// TIA Portal V16 export
// export: Created 2023-02-01T15:24:13.3591852Z, ExportSetting WithDefaults, DisplayName Totally Integrated Automation Portal, DisplayVersion V16 Update 3, DisplayName TIA Portal Version Control Interface, DisplayVersion V16 Update 2, DisplayName TIA Portal Openness, DisplayVersion V16 Update 3, DisplayName STEP 7 Professional, DisplayVersion V16 Update 3, DisplayName STEP 7 Safety, DisplayVersion V16, DisplayName WinCC Professional, DisplayVersion V16 Update 3
FUNCTION "FC11101_StdDevValveBi" : Void   // FC11101, LAD
TITLE = Standard Module [DEVICE DRIVER] — Bistable Valve
{ S7_Optimized_Access := 'TRUE' }
AUTHOR : M_Gledhill
FAMILY : DeviceDriver
NAME : StdDevValveBi
VERSION : 0.8
// PRACTICAL SERIES AUTOMATION LIBRARY (PAL)   —   COPYRIGHT 2020 – M. GLEDHILL (MIT LICENCE)
//                   ———— ◆ ————
// FULL ONLINE DOCUMENTATION IS AVAILABLE AT: https://practicalseries.com/2001-pal/index.html
// stored: AutoNumber false, IsIECCheckEnabled true, SetENOAutomatically false, UDAEnableTagReadback false
   VAR_INPUT
      SYS_SIGNALS : "UT21000_Dy_SysSignals";   // Common system signals — logic and timing signals
      FBK_OPEN : Bool;   // Positive open position feedback (1 = valve open, 0 = valve not open)
      FBK_CLOSED : Bool;   // Positive closed position feedback (1 = valve closed, 0 = valve not closed)
      EXT_FAULT : Bool;   // Device external fault signal (1 = fault, 0 = healthy)
      E_STOP : Bool;   // Safety (E-STOP) signal (1 = ESTOP active, 0 = healthy)
      TRIP : Bool;   // Interlock (TRIP) signal (1 = TRIP active, 0 = healthy)
      INTERLOCK : Bool;   // Interlock (INTERLOCK) signal (1 = INTERLOCK active, 0 = healthy)
      PERMISSIVE : Bool;   // Interlock (PERMISSIVE) signal (1 = PERMISSIVE active, 0 = healthy)
      STATIC_DATA : "UT11101_St_DevValveBi";   // Static data storage (UDT)
   END_VAR
   VAR_OUTPUT
      OPEN_CMD : Bool;   // Valve open signal (1 = open the valve, 0 = no action)
      CLOSE_CMD : Bool;   // Valve close signal (1 = close the valve, 0 = no action)
   END_VAR
   VAR_IN_OUT
      DYNAMIC_DATA : "UT31101_Dy_DevValveBi";   // Dynamic data storage (UDT)
   END_VAR
   VAR_TEMP
      revInfo : "UT01000_St_SysRevision";   // Revision information for this block
      licInfo : "UT01001_St_SysLicence";   // Licensing information for this block
      calClosedElapsedTime : Real;   // Calculation - Derived closed signal elapsed time limit
      calOpenElapsedTime : Real;   // Calculation - Derived open signal elapsed time limit
      wrkOpen : Bool;   // Working - open position feedback signal (actual or derived)
      wrkClosed : Bool;   // Working - closed position feedback signal (actual or derived)
      wrkCtrlPriority40 : Bool;   // Working - priority 40 condition controls the valve
      wrkCtrlPriority30 : Bool;   // Working - priority 30 condition controls the valve
      wrkCtrlPriority20 : Bool;   // Working - priority 20 condition controls the valve
      wrkCtrlPriority10 : Bool;   // Working - priority 10 condition controls the valve
      wrkCtrlPriority00 : Bool;   // Working - priority 00 condition controls the valve
      wrkCtrlAutManOpCl : Bool;   // Working - consolidated auto/manual open or close request
      wrkTimeFbkOpenDer : Real;   // Working - value of opening timer before derived open feedback
      wrkTimeFbkClosedDer : Real;   // Working - value of closing timer before derived closed feedback
      wrkInt : Int;   // Working - storage area (integer)
      wrkReal : Real;   // Working - storage area (Real)
      wrkDInt : DInt;   // Working - storage area (double integer)
   END_VAR
   VAR CONSTANT
      k_TIME_OP_MIN : Real := 0.21;   // Minimum value for the valve operation timer
      K_TIME_SIM_MIN : Real := 0.21;   // Minimum value for the simulation operation timer
   END_VAR
   VAR_TEMP   // added for the SCL form of the ladder/FBD networks
      _w1 : Bool;
      _w2 : Bool;
      _w3 : Bool;
   END_VAR
BEGIN

REGION Network 1: Block description — Sections 1 to 2
   // ▄▄▄▄▄▄▄▄▄▄▄▄▄▄▄▄▄▄▄▄▄▄▄▄▄▄▄▄▄▄▄▄▄  ＳＴＡＮＤＡＲＤ  ▄▄ 
   // 
   // 
   // TITLE:    DEVICE DRIVER — BISTABLE VALVE
   // 
   // 
   // ▀▀▀▀▀▀▀▀▀▀▀▀▀▀▀▀▀▀▀▀▀▀▀▀▀▀▀▀▀▀▀▀▀▀▀▀▀▀▀▀▀▀▀▀ 
   // 
   // ┌──────────────────────────────────────────┐
   // │                                          │
   // │          FC11101 — SOFTWARE MODULE DESIGN SPECIFICATION (SMDS)            │
   // │                                          │
   // │      The PDF version of the SMDS for this module is available online here:        │
   // │              https://psop.uk/pal-smds-fc11101-p               │
   // │                                          │
   // │      It is also available as part of the Project User Defined Documentation,      │
   // │      it can be accessed by selecting this module in the Project Tree          │
   // │      (on the left) and pressing SHIFT+F1                        │
   // │                                          │
   // └─────────────────────────────────────── ʷᴵᴰ⁻ᶜᵇᵃ ┘
   // 
   // FC11101_StdDevValveBi controls the operation of a bistable valve configured with either open, 
   // closed, both open and closed or no position feedback (depending on the valve type).
   // 
   // The module supports automatic and manual control and can be configured with simulation 
   // mode to allow the valve limit switch signals to be overwritten and set to follow the demand 
   // position.
   // 
   // The module can be configured to either de-energise the outputs when the valve reaches the 
   // demanded position, or maintain the outputs when position is reached.
   // 
   // The module generates fault logic for the valve that will trigger specific alarms depending on the 
   // fault in question. The alarms within this block are: 
   // 
   // 
   //    •   Failed to Open 
   // 
   //    •   Failed to Close 
   // 
   //    •   Failed while Open
   // 
   //    •   Failed while Closed
   // 
   //    •   External Fault 
   // 
   // Separate operation times for opening and closing can be defined. 
   // 
   // The valve module supports all forms of interlock, permissive and trip signals, and emergency 
   // stop signals. The module has the conditional facility to allow the operator to bypass interlocks, 
   // permissive and trip conditions.
   // 
   // Various status signals are generated for supervisory systems:
   // 
   //    •   Closed
   // 
   //    •   Closing
   // 
   //    •   Open
   // 
   //    •   Opening
   // 
   //    •   Fault
   // 
   // The module also generates status signals for the selected operating modes and conditions.
   // 
   // 
   // 
   // ▄▄▄▄▄▄▄▄▄▄▄▄▄▄▄▄▄▄▄▄▄▄▄▄▄▄▄▄▄▄▄▄▄▄▄▄▄▄▄▄▄▄▄▄
   // 1.     BLOCK TECHNICAL SUMMARY
   // 
   // 
   //  ――――――――――――――――――――――――――――――――――――――――――
   //  NOMENCLATURE & ADDRESSING
   //  ――――――――――――――――――――――――――――――――――――――――――
   //  BLOCK TITLE         Bistable Valve
   //  BLOCK FUNCTION GROUP    Device Driver 
   //  BLOCK ADDRESS       FC11101
   //  BLOCK SYMBOL        FC11101_StdDevValveBi
   //  BLOCK USER ID         StdDevValveBi
   // 
   //  ――――――――――――――――――――――――――――――――――――――――――
   //  BLOCK TYPE & USAGE
   //  ――――――――――――――――――――――――――――――――――――――――――
   //  BLOCK TYPE         Function (FC)
   //  BLOCK NUMBER        11101
   //  LANGUAGE           LAD
   //  OPTIMISED ACCESS     Yes
   //  PAL USAGE TYPE       Standard block
   // 
   //  ――――――――――――――――――――――――――――――――――――――――――
   //  METRICS
   //  ――――――――――――――――――――――――――――――――――――――――――
   //  EXECUTION TIME       81.3 μs¹
   //  LOAD MEMORY       113.1 kB
   //  WORK MEMORY           2.5 kB  
   //  ――――――――――――――――――――――――――――――――――――――――――
   //                ¹ Measured on: CPU-1515-2PN (order no. 6ES7512-2AM02-0AB0) 
   //                             https://psop.uk/pal-ds-cpu1515
   // 
   // 
   // 
   // ▂▂▂▂▂▂▂▂▂▂▂▂▂▂▂▂▂▂▂▂▂▂▂▂▂▂▂▂▂▂▂▂▂▂▂▂▂▂▂▂▂▂▂▂
   // 1.1      Additional document references
   // 
   // 
   // Only those documents specified in OB1 (section DOCUMENT REFERENCES) are listed within this 
   // block. There are no additional document references.
   // 
   //                ━━━   ⬙⬙⬙⬙⬙⬙   ━━━
   // 
   // 
   // 
   // ▄▄▄▄▄▄▄▄▄▄▄▄▄▄▄▄▄▄▄▄▄▄▄▄▄▄▄▄▄▄▄▄▄▄▄▄▄▄▄▄▄▄▄▄
   // 2.     FUNCTIONAL DESCRIPTION
   // 
   // 
   // FC11101 is the Bistable Valve block, it is a comprehensive block designed to operate and monitor 
   // a standard bistable valve. 
   // 
   // 
   // 
   // ▂▂▂▂▂▂▂▂▂▂▂▂▂▂▂▂▂▂▂▂▂▂▂▂▂▂▂▂▂▂▂▂▂▂▂▂▂▂▂▂▂▂▂▂
   // 2.1     Defining a bistable valve
   // 
   // 
   // A bistable valve is any valve that has two signals to make it change state; it has two mutually 
   // exclusive output signals: an OPEN_CMD output that must be energised to drive the valve to the 
   // open position and a CLOSE_CMD output that must be energised to drive the valve to the closed 
   // position.
   // 
   // To open the valve the OPEN_CMD signal must be energised and the CLOSE_CMD signal 
   // deenergised. When the valve reaches the opened position, both signals will be deenergised² and 
   // the valve will remain in the opened state (it is stable in this condition and does not require any 
   // signal to maintain it in this state, if there were a power failure the valve would remain opened).
   // 
   // To close the valve the CLOSE_CMD signal must be energised and the OPEN_CMD signal 
   // deenergised. When the valve reaches the closed position, both signals will again be 
   // deenergised² and the valve will remain in the closed state (again the valve is stable in this 
   // condition and does not require any signal to maintain it in this state, if there were a power failure 
   // the valve would remain closed).
   // 
   // This is said to be a bistable device because once it is in a particular state, it does not (generally) 
   // require any signal to be energised to maintain that state.
   // 
   // ――――――――――
   // ²         The module can also be configured to maintain the appropriate output signal once 
   //      the required state is achieved (see § 3.2.1).
   // ――――――――――
   // 
   // 
   // 
   // ▂▂▂▂▂▂▂▂▂▂▂▂▂▂▂▂▂▂▂▂▂▂▂▂▂▂▂▂▂▂▂▂▂▂▂▂▂▂▂▂▂▂▂▂
   // 2.1.1     Comparison with an isolating valve
   // 
   // 
   // In many ways a bistable valve is very similar to an isolating valve (controlled by FC11001), it 
   // generally has only two states (it is either opened or closed); however, because the bistable valve 
   // is electrically driven (usually by a motor), if the driving signals are removed while the valve is in 
   // transit (say via an emergency stop being activated), the valve will simply stop in its current 
   // (intermediate) position and remain there until a driving signal is re-applied. This situation is 
   // discussed in §§ 2.3.1 and 3.4.1.
   // 
   // Additionally, because the bistable valve is stable in both the open and closed positions, the 
   // bistable valve does not have the normally open and normally closed³  types available to an 
   // isolating valve. A Bistable valve does not return to a specific state if power is removed from the 
   // actuator; it simply remains in its current state (even if this is an indeterminate state).
   // 
   // ――――――――――
   // ³         For an isolating valve, normally closed refers to a valve that is deenergised in the 
   //      closed state and will open when an energising signal is applied. A normally open 
   //      valve operates in the reverse arrangement, the valve is open in the deenergised 
   //      state and will only close when the energising signal is present. Normally open valves 
   //      are used in fail-safe applications where a power failure causes the valve to open by 
   //      default, usually to vent pressure or release some other motive force from the vessel 
   //      to which it is connected.
   // ――――――――――
   // 
   // 
   // 
   // 
   // ▂▂▂▂▂▂▂▂▂▂▂▂▂▂▂▂▂▂▂▂▂▂▂▂▂▂▂▂▂▂▂▂▂▂▂▂▂▂▂▂▂▂▂▂
   // 2.1.2     Valve operating times
   // 
   // 
   // A bistable valve, will move from its closed state to its open state when the OPEN_CMD signal is 
   // applied; this transition will occur in a specified time (the time taken will depend on the size and 
   // operating mechanism within the valve itself), this is referred to as the opening operation time.
   // 
   // Similarly, the transition from open to closed will occur when the CLOSE_CMD signal is applied, 
   // and again, this will occur in a specified time. This is referred to as the closing operation time. 
   // 
   // The opening and closing times can be different for a given valve. 
   // 
   // Collectively, the opening and closing times are referred to as the operating times (sometimes 
   // operation times) of the valve.
   // 
   // The maximum opening and closing times for a valve are generally given as part of the 
   // specification for the valve itself.
   // 
   // If a valve does not reach the required state within the specified maximum operating times, the 
   // valve is generally considered to be in a fault condition (either failed to open or failed to close 
   // depending on the action being undertaken).
   // 
   // 
   // 
   // ▂▂▂▂▂▂▂▂▂▂▂▂▂▂▂▂▂▂▂▂▂▂▂▂▂▂▂▂▂▂▂▂▂▂▂▂▂▂▂▂▂▂▂▂
   // 2.1.3     Valve position feedback arrangements
   // 
   // 
   // Bistable valves can be equipped with limit switch signals that positively identify the current 
   // position of the valve. There are four combinations of limit switches:
   // 
   //    1.  No limit switches         There is no positive indication of the current state 
   //                      of the valve, it is assumed to be in the expected 
   //                      state.
   // 
   //    2.  Closed limit switch only       Positive indication is given for the closed state 
   //                      only. The valve is assumed to be open (after a 
   //                      predetermined time) if the closed signal is 
   //                      inactive
   // 
   //    3.  Open limit switch only      Positive indication is given for the open state 
   //                      only. The valve is assumed to be closed (after a 
   //                      predetermined time) if the open signal is 
   //                      inactive.
   // 
   //    4.  Open and closed limit switches    Positive indication is given for both states. 
   //                      This allows the true state of the valve to be 
   //                      determined under all circumstances.
   // 
   // Note:    Positive indication of a valve state need not be determined by a limit switch 
   //      (though this is by far the most common arrangement), it could for example, be 
   //      determined by some process value: if a flow is detected after the opening of a valve, 
   //      for example.
   // 
   //      In practice, limit switches are the preferred mechanism for the positive indication 
   //      of a given valve state.
   // 
   // Where a limit switch is absent, the valve is assumed to have reached the correct position when 
   // the relevant operation time has counted for an adjustable percentage of its maximum operating 
   // time.
   // 
   // The valve can be configured to “run-on” for a specified time after the demanded position has been 
   // achieved (i.e. the block will maintain the driving signal for a time period after the limit switch is 
   // activated to ensure the valve is firmly in position).
   // 
   // The valve can also be configured to maintain either the OPEN_CMD signal or the CLOSE_CMD 
   // signal permanently once the valve has reached the desired position; i.e. the OPEN/CLOSE_CMD 
   // signals do not deenergise when the valve has reached the correct position. 
   // 
   // 
   // 
   // ▂▂▂▂▂▂▂▂▂▂▂▂▂▂▂▂▂▂▂▂▂▂▂▂▂▂▂▂▂▂▂▂▂▂▂▂▂▂▂▂▂▂▂▂
   // 2.2     Module operation
   // 
   // 
   // FC11101 is used to control (operate) a bistable valve, the module also monitors the various 
   // configurations of valve position feedback signals to determine if the valve is in a fault condition.
   // 
   // The module will drive the valve to the requested state by energising and deenergising two 
   // separate (mutually exclusive) digital signals (usually digital output signals), one signal to open 
   // the valve and one to close it.
   // 
   // These digital output signals can be configured to either deenergise when the valve reaches the 
   // required state (with a configurable run-on time) or to remain energised when the final state is 
   // reached.
   // 
   // If the requested state signal changes (either from closed to open, or from open to closed), the 
   // module will start either an opening operation timer (request has changed from closed to open) 
   // or a closing operation timer (request has changed from open to closed); these timers can have 
   // different values.
   // 
   // The valve will be expected to reach the requested state before the relevant operation timer 
   // expires; if it does not, the valve will enter a fault state and an appropriate alarm will be generated 
   // when the operation timer expires.
   // 
   // Once the valve has reached its requested state, the operation time will reset and the module 
   // will continue to monitor the state of the valve. 
   // 
   // If the request signal changes whilst the valve is in the process of changing state (e.g. the valve 
   // is requested to change from closed to open and whilst the opening operation timer is running, 
   // the request is changed back to closed), the running operation timer will be reset and the 
   // operation timer for the second request will start from its specified value. I.e. no allowance is 
   // made for how far the valve may have moved following the first request change.
   // 
   // If the valve is stable, in a given state (i.e. is not in the process of changing state) and the valve 
   // position signals no longer match the required state (e.g. the valve had correctly opened, but at 
   // some time after this, the open position feedback is lost), the valve will instantly generate an 
   // alarm condition.
   // 
   // 
   // 
   // ▂▂▂▂▂▂▂▂▂▂▂▂▂▂▂▂▂▂▂▂▂▂▂▂▂▂▂▂▂▂▂▂▂▂▂▂▂▂▂▂▂▂▂▂
   // 2.3     Safety and interlocks
   // 
   // 
   // The module, optionally, accommodates a single safety signal (emergency stop), and the 
   // standard arrangement of up to three interlock signals (interlock, permissive and trip) as follows:
   // 
   // 
   // 
   // ▂▂▂▂▂▂▂▂▂▂▂▂▂▂▂▂▂▂▂▂▂▂▂▂▂▂▂▂▂▂▂▂▂▂▂▂▂▂▂▂▂▂▂▂
   // 2.3.1     Safety (emergency stop) signal
   // 
   // 
   // Safety or emergency stop signals are hardwired signals that remove power from a device forcing 
   // it to a safe state. Such signals act independently of the software (the pressing of an emergency 
   // stop button will physically remove power from the affected devices).
   // 
   // In the case of a bistable valve, the removing of the power under emergency stop conditions, 
   // simply deenergises both outputs leaving the valve in its current state¹: if the valve were already 
   // open, it would remain open, similarly if the valve were closed, it would remain closed.
   // 
   // The leads to the question, what happens if an emergency stop activates when the valve is 
   // changing state? The answer is that the valve simply stops where it is in mid-transition (in some 
   // indeterminate, intermediate state between open and closed). To accommodate this condition, 
   // the active operation timer will simply pause at its elapsed value (the valve will remain in either 
   // the opening or closing state) until the emergency stop condition is removed, at this point, the 
   // operation timer will continue from its last elapsed value .
   // 
   // Note:    The resumption of the operation timer can be delayed by a recovery time, this is
   //      to allow the physical aspects of the valve itself to reset and resume operation 
   //      (e.g. to allow the valve motor to ramp to the correct speed &c.), this recovery time 
   //      is configurable.
   // 
   // The emergency stop signal passed to the module is used to allow the condition of the valve to 
   // be correctly interpreted within the software under emergency stop conditions.
   // 
   // The presence of an emergency stop signal is indicated via the block icon status signals generated 
   // by the module (see §§ 2.7 and 4.2).
   // 
   // Emergency stop signals cannot be bypassed under any circumstances (cf. interlock signals, 
   // below).
   // 
   // ――――――――――
   // ¹         This is unlike the isolating valve of FC11001; the isolating valve returns to a particular 
   //      state (either open or closed depending on the normally open/closed arrangement of 
   //      the valve). By comparison, the bistable simply stops in the condition it is in.
   // ――――――――――
   // 
   // 
   // 
   // ▂▂▂▂▂▂▂▂▂▂▂▂▂▂▂▂▂▂▂▂▂▂▂▂▂▂▂▂▂▂▂▂▂▂▂▂▂▂▂▂▂▂▂▂
   // 2.3.2     Interlock signals
   // 
   // 
   // There are three types of interlock signal:
   // 
   //    1.  Interlock
   //      A simple interlock that is active whenever a set of conditions is true; if active, it will 
   //      force the devices to a specified state.
   // 
   // 
   //    2.  Permissive
   //      Designates a specified “permitted” state for the device. A permissive interlock takes 
   //      no action if the device is in the non-permitted state, but once the device changes to 
   //      the permitted state, it will be prevented from changing back to the non-permitted state 
   //      (e.g. if the permitted state was closed and the valve was currently open when the 
   //      permissive signal activated, it would not force the valve to close, but once it was 
   //      closed, it would prevent it from re-opening).
   // 
   //    3.  Trip
   //      A latching interlock, it activates whenever a set of events are true (like an interlock), 
   //      but will not deactivate until the triggering conditions are removed and a reset signal 
   //      has been given (effectively a latching interlock); if active, it will force the device to a 
   //      specified state.
   // 
   // Note:    The trip reset signal is handled by the trip logic, the valve module will simply respond 
   //      to the presence or absence of a trip signal.
   // 
   // Each type of interlock has its own individual signal passed to the module (three signals in total).
   // 
   // Interlock signals can be optionally bypassed (effectively disabled) under specific, manually 
   // selected operations.
   // 
   // 
   // 
   // ▂▂▂▂▂▂▂▂▂▂▂▂▂▂▂▂▂▂▂▂▂▂▂▂▂▂▂▂▂▂▂▂▂▂▂▂▂▂▂▂▂▂▂▂
   // 2.3.3     Priority of safety and interlock signals
   // 
   // 
   // The presence of any interlock stop signal is indicated via the block icon status signals generated 
   // by the module (see § 4). The priority order of the various types of interlock (if more than one is 
   // active at the same time) is as follows:
   // 
   // 
   //  ――――――――――――――――――――――――――――――――――――――――――
   //  SIGNAL TYPE        PRIORITY        CAN BE BYPASSED
   //  ――――――――――――――――――――――――――――――――――――――――――
   //  Emergency Stop         High               NO
   //  Trip             ↑              YES
   //  Interlock             ↑              YES
   //  Permissive          Low               YES
   //  ――――――――――――――――――――――――――――――――――――――――――
   //  High priority signal take precedence over lower priority signals.
   // 
   // 
   // 
   // ▂▂▂▂▂▂▂▂▂▂▂▂▂▂▂▂▂▂▂▂▂▂▂▂▂▂▂▂▂▂▂▂▂▂▂▂▂▂▂▂▂▂▂▂
   // 2.4     Alarms and warnings
   // 
   // 
   // The module can generate up to five distinct alarms:
   // 
   // 
   //    1.  FAILED TO OPEN
   //      Indicates that the valve did not open when requested to do so. The alarm is generated 
   //      when the opening operation timer expires without the corresponding position feedback 
   //      activating
   // 
   //    2.  FAILED TO CLOSE
   //      Indicates that the valve did not close when requested to do so. The alarm is generated 
   //      when the closing operation timer expires without the corresponding position feedback 
   //      activating
   // 
   // 
   //    3.  FAILED WHILE OPEN
   //      Indicates that the valve opened correctly, but then at some later point, the position 
   //      feedback signals, indicating the open state of the valve, were lost.
   // 
   //    4.  FAILED WHILE CLOSED
   //      Indicates that the valve closed correctly, but then at some later point, the position 
   //      feedback signals, indicating the closed state of the valve, were lost.
   // 
   // 
   //    5.  EXTERNAL FAULT
   //      External fault is a separate (and optional) hardwired signal from the valve that 
   //      indicates the valve itself has detected a problem (e.g. a trip signal from a 
   //      motorised valve)
   // 
   // The module does not generate any warnings.
   // 
   // 
   // 
   // ▂▂▂▂▂▂▂▂▂▂▂▂▂▂▂▂▂▂▂▂▂▂▂▂▂▂▂▂▂▂▂▂▂▂▂▂▂▂▂▂▂▂▂▂
   // 2.4.1     Alarm — Failed to open/close
   // 
   // 
   // Failed to open and failed to close alarms are generated if the valve is required to change state 
   // and fails to do so within the time set by the relevant operation timer.
   // 
   // For example, if the valve were in a closed state and was requested to open, the failed to open 
   // alarm would be generated if the valve had not received positive indication that the valve was 
   // correctly open (from the valve limit switches) by the time the opening operation timer expired.
   // 
   // If the valve is not equipped with any limit switches, then there are no circumstances under 
   // which the failed to open and failed to close alarms can be generated (the valve is always 
   // assumed to operate correctly and be in the required position).
   // 
   // 
   // 
   // ▂▂▂▂▂▂▂▂▂▂▂▂▂▂▂▂▂▂▂▂▂▂▂▂▂▂▂▂▂▂▂▂▂▂▂▂▂▂▂▂▂▂▂▂
   // 2.4.2     Alarm — Failed while open/closed
   // 
   // 
   // Failed while open and failed while closed are generated if the valve is in a steady state (not in 
   // the process of changing from open to closed or vice versa) and the positive indication of the 
   // valve position changes to indicate the steady state position has changed.
   // 
   // An example would be for a normally closed valve, with both open and closed limit switches, 
   // to be in the open (energised) state, where the open limit is active and closed limit is inactive 
   // (positively indicating the valve is open). If the power to the valve failed (a blown fuse or broken 
   // wire, for example), the valve would deenergise and return to the closed state and this would be 
   // reflected in the state of the limit switches. The module, knowing nothing of the power failure, 
   // would expect the valve to still be open and would instantly generate a failed while open alarm.
   // 
   // If the valve is not equipped with any limit switches, then there are no circumstances under which 
   // the failed while open and failed while closed alarms can be generated (the valve is always 
   // assumed to operate correctly and be in the required position).
   // 
   // 
   // 
   // ▂▂▂▂▂▂▂▂▂▂▂▂▂▂▂▂▂▂▂▂▂▂▂▂▂▂▂▂▂▂▂▂▂▂▂▂▂▂▂▂▂▂▂▂
   // 2.4.3     Alarm — External fault
   // 
   // 
   // The external fault alarm is activated whenever the external fault signal provided to the module 
   // is active. The external fault signal is an optional signal that indicates that the valve itself is 
   // experiencing a problem. The signal is more commonly associated with motorised valves where 
   // thermal overload signals are used to indicate that the valve motor has experienced a fault, 
   // it could also be used to indicate the loss of pneumatic pressure for pneumatic solenoid valves.
   // 
   // 
   // 
   // ▂▂▂▂▂▂▂▂▂▂▂▂▂▂▂▂▂▂▂▂▂▂▂▂▂▂▂▂▂▂▂▂▂▂▂▂▂▂▂▂▂▂▂▂
   // 2.4.4     Resetting alarm conditions
   // 
   // 
   // The four alarms derived from valve position feedback signals:
   // 
   //    1.  FAILED TO OPEN
   // 
   //    2.  FAILED TO CLOSE
   // 
   //    3.  FAILED WHILE OPEN
   // 
   //    4.  FAILED WHILE CLOSED
   // 
   // Are latching alarms, if the alarm conditions occur, the valve will be placed in a fault condition 
   // (see § 2.5) and will no longer be operable, the valve will remain in a deenergised condition until 
   // the fault is corrected.
   // 
   // The alarm conditions are only reset when the module receives a RESET command (usually 
   // from the operator).
   // 
   // The fifth alarm:
   // 
   //    5.  EXTERNAL FAULT
   // 
   // Is a non-latching alarm that is reset automatically whenever the external fault signal is 
   // deactivated. It should be noted however, that the cause of the external fault (say a thermal 
   // overload) may itself, require some form of manual or physical reset, before the fault condition 
   // is removed.
   // 
   // 
   // 
   // ▂▂▂▂▂▂▂▂▂▂▂▂▂▂▂▂▂▂▂▂▂▂▂▂▂▂▂▂▂▂▂▂▂▂▂▂▂▂▂▂▂▂▂▂
   // 2.5     Fault conditions
   // 
   // 
   // The valve is in a fault condition if any alarm conditions is active:
   // 
   //    1.  FAILED TO OPEN
   // 
   //    2.  FAILED TO CLOSE
   // 
   //    3.  FAILED WHILE OPEN
   // 
   //    4.  FAILED WHILE CLOSED
   // 
   //    5.  EXTERNAL FAULT
   // 
   // A valve cannot operate if any fault condition is active and it will return to its deenergised state.
   // 
   // For a normally closed valve, the deenergised state is closed and for a normally open valve, 
   // the deenergised state is open.
   // 
   // A valve that is in a fault state will ignore any request that would move it to an energised state, 
   // irrespective of the source of the command: automatic operation, manual operation or even an 
   // interlock condition.
   // 
   // 
   // The valve will remain in a fault state until all alarms have been reset, in the case of the four limit 
   // switch derived alarms the module must receive a RESET command (see § 2.4.4) to remove the 
   // alarms, and consequently, the fault conditions.
   // 
   // The EXTERNAL FAULT alarm is a non-latching alarm that is reset automatically whenever the 
   // external fault signal is deactivated, consequently, the fault state will automatically reset when 
   // the external fault signal deactivates.
   // 
   // It should be noted however, that the cause of the external fault (say a thermal overload) may 
   // itself, require some form of manual or physical reset, before the fault condition is removed.
   // 
   // 
   // 
   // ▂▂▂▂▂▂▂▂▂▂▂▂▂▂▂▂▂▂▂▂▂▂▂▂▂▂▂▂▂▂▂▂▂▂▂▂▂▂▂▂▂▂▂▂
   // 2.6     Operating modes
   // 
   // 
   // The module supports the following optional modes of operation:
   // 
   //    •   Automatic/manual mode (allows the operator to take manual control of the valve 
   //      and open or close it irrespective of the control system requirements)
   // 
   //    •   Interlock bypass mode (allows the operator to override permissive, interlock and 
   //      trip signals
   // 
   //    •   Simulation mode (allows the operator to override the current instrument position 
   //      feedback signals  simulated values)
   // 
   //    •   Remote/local/all selection (allows control of the instrument to be restricted to a 
   //      specific SCADA/HMI device) 
   // 
   //    •   Faceplate disabled (informs the supervisory system not to display any faceplates 
   //      for the device, preventing graphical operator selections)
   // 
   // 
   // 
   // ▂▂▂▂▂▂▂▂▂▂▂▂▂▂▂▂▂▂▂▂▂▂▂▂▂▂▂▂▂▂▂▂▂▂▂▂▂▂▂▂▂▂▂▂
   // 2.6.1     Automatic and manual control modes
   // 
   // 
   // By default, the module will be in automatic mode; this means that any open or close instruction 
   // received by the module from the control software (continuous or sequential control) will cause 
   // the valve to adopt the requested state (if the valve is not in fault and is free of interlock and 
   // safety conditions).
   // 
   // If the module is switched to manual mode, the automatic control signals will be ignored and the 
   // module will adopt the state required by the manual request signals set by the operator 
   // (again, the valve must not be in fault and must be free of interlock and safety conditions).
   // 
   // Selecting automatic or manual mode is an operator action and can be implemented at any time. 
   // Changing from automatic mode to manual mode is a bumpless operation, in which the initial 
   // manual state of the valve is set to match the current automatic state. For example, if a valve 
   // were open under automatic control, switching the valve to manual would cause the initial 
   // manual state to be set to open (matching the automatic state), ensuring that the valve does not 
   // initially change state when changing to manual mode.
   // 
   // Once manual mode is established, the operator is free to open and close the valve as required.
   // 
   // There is no bumpless transfer back to automatic mode, the valve will simply adopt the state 
   // required by the control software.
   // 
   // Interlocks and safety signals operate in exactly the same way for a valve in manual mode 
   // as they do for a valve in automatic mode and will take priority over any command issued in either 
   // automatic or manual mode.
   // 
   // 
   // 
   // ▂▂▂▂▂▂▂▂▂▂▂▂▂▂▂▂▂▂▂▂▂▂▂▂▂▂▂▂▂▂▂▂▂▂▂▂▂▂▂▂▂▂▂▂
   // 2.6.2     Interlock bypass mode
   // 
   // 
   // Interlock bypass mode allows the three interlock types (trip, interlock and permissive) to be 
   // overridden (bypassed) by the operator.
   // 
   // If bypass mode is activated, any interlock signal will be ignored by the module.
   // 
   // Bypass mode is an entirely manual operation that can only be initiated by an operator, usually 
   // via a supervisory system (SCADA or HMI).
   // 
   // 
   // 
   // ▂▂▂▂▂▂▂▂▂▂▂▂▂▂▂▂▂▂▂▂▂▂▂▂▂▂▂▂▂▂▂▂▂▂▂▂▂▂▂▂▂▂▂▂
   // 2.6.3     Simulation mode
   // 
   // 
   // The module can be switched to a simulation mode, under which any positive position feedback 
   // signals from valve limit switches are replaced by simulated signals selected by the operator. 
   // Simulation mode can be used during testing and can also be applied in a process environment 
   // if a fault condition is detected within the valve.
   // 
   // The operator can select any one of the following possible simulation arrangements (only one 
   // can be active at any given time):
   // 
   // 
   //    •   Follow demand    The simulation will generate open and closed signals that 
   //                 match the requested state of the valve
   // 
   //    •   Open          The simulation will generate signals to give a permanently 
   //                 open state for the valve, irrespective of any valve state 
   //                 request (allows failed open conditions to be simulated)
   // 
   //    •   Closed           The simulation will generate signals to give a permanently 
   //                 closed state for the valve, irrespective of any valve state 
   //                 request (allows failed closed conditions to be simulated)
   //                 request (allows failed open conditions to be simulated)
   // 
   //    •   No limits       No position feedback signals will be simulated
   // 
   // Simulation mode is a manual operation that can only be initiated by an operator.
   // 
   // 
   // 
   // ▁▁▁▁▁▁▁▁▁▁▁▁▁▁▁▁▁▁▁▁▁▁▁▁▁▁▁▁▁▁▁▁▁▁▁▁▁▁▁▁▁▁▁▁
   // 2.6.4     Remote/local/all mode
   // 
   // Remote and local operating modes refer to the device that has control of the module; where 
   // a plant has more than one SCADA/HMI, say a SCADA in a remote control room and a field 
   // mounted HMI local to the device, it is possible to restrict the operator control of the module to 
   // one, or the other, or both supervisor systems as follows
   // 
   //    •   Remote Only the remote system in the control room can control the device
   // 
   //    •   Local     A local system has taken control of the device and the remote system can 
   //            no longer issue commands to it
   // 
   //    •    All    Any system can control the device
   // 
   // The default arrangement if for all systems to have access to the device.
   // 
   // 
   // 
   // ▁▁▁▁▁▁▁▁▁▁▁▁▁▁▁▁▁▁▁▁▁▁▁▁▁▁▁▁▁▁▁▁▁▁▁▁▁▁▁▁▁▁▁▁
   // 2.6.5     Faceplate disabled mode
   // 
   // Prevents the supervisory system from displaying the faceplate from which the above options are 
   // selected. If the faceplate is disabled, the operator will not be able to select or change any of the 
   // various operating modes.
   // 
   // 
   // 
   // ▁▁▁▁▁▁▁▁▁▁▁▁▁▁▁▁▁▁▁▁▁▁▁▁▁▁▁▁▁▁▁▁▁▁▁▁▁▁▁▁▁▁▁▁
   // 2.7      Supervisory system interface
   // 
   // See the online documentation for this block — select the block in the project tree and press:
   //      SHIFT + F1 or follow the link: https://psop.uk/pal-smds-fc11101-p 
   // 
   // The supervisory system interface is available in sections 2.5 and 4 of the online SMDS 
   // document.
   // 
   //                ━━━   ⬙⬙⬙⬙⬙⬙   ━━━
END_REGION

REGION Network 2: Block description — Section 3 to 3.2.5
   // ▄▄▄▄▄▄▄▄▄▄▄▄▄▄▄▄▄▄▄▄▄▄▄▄▄▄▄▄▄▄▄▄▄▄▄▄▄▄▄▄▄▄▄▄
   // 3.     DETAILED BLOCK DESCRIPTION
   // 
   // 
   // This module, FC11101_StdDevValveBi uses user data types to provide the primary interface to 
   // the module, it also uses direct digital signals to provide an interface for the position feedback 
   // signals and for the fault, safety and interlock signals. It also has a single output signal used to 
   // operate the valve. 
   // 
   // These are the formal module parameters: 
   // 
   //  ――――――――――――――――――――――――――――――――――――――――――
   //  PARAM         FUNCTION                    TYPE      IN-OUT 
   //  ――――――――――――――――――――――――――――――――――――――――――
   //  SYS_SIGNALS      Common system signals              UT21000    In
   //           logic and timing signals for parametric access
   // 
   //  FBK_OPEN     Optional open state positive feedback        Bool      In
   //           (1 = open, 0 = not open) If not required, set 
   //           permanently to _False
   // 
   //  FBK_CLOSED    Optional closed state positive feedback        Bool      In
   //           (1 = closed 0 = not closed) If not required, set 
   //           permanently to _False
   // 
   //  EXT_FAULT     Optional external fault signal for the device     Bool      In
   //           (1 = fault, 0 = healthy). If not required, set 
   //           permanently to _False
   // 
   //  E_STOP        Optional emergency stop (safety) signal        Bool      In
   //           (1 = emergency stop active, 0 = healthy) If not 
   //           required, set permanently to _False
   // 
   //  TRIP        Optional trip signal                  Bool      In
   //           (1 = trip condition active, 0 = healthy) If not 
   //           required, set permanently to _False
   // 
   //  INTERLOCK     Optional interlock signal               Bool      In
   //           (1 = interlock condition active, 0 = healthy) If 
   //           not required, set permanently to _False
   // 
   //  PERMISSIVE      Optional permissive signal             Bool      In
   //           (1 = permissive condition active, 0 = healthy) 
   //           If not required, set permanently to _False
   // 
   //  STATIC_DATA     Data structure that holds the configuration data     UT11101    In
   //           for the device (limit switch, timer presets 
   //           and interlock configuration &c.)
   // 
   //  DYNAMIC_DATA      Data structure that holds the live data for the       UT31101    InOut
   //           device (its mode, status, messages and 
   //           other dynamic information)
   // 
   //  OPEN_CMD       Output to drive the valve to an open state    Bool      Out
   //           (1 = Open valve, 0 = no action)
   // 
   //  CLOSE_CMD     Output to drive the valve to a closed state       Bool      Out
   //           (1 = Close valve, 0 = no action)
   //  ――――――――――――――――――――――――――――――――――――――――――
   // 
   // FBK_OPEN, FBK_CLOSED and EXT_FAULT parameters are input signals provided directly from the 
   // device itself (via digital input cards). 
   // 
   // The E-STOP parameter is the interface to any safety signal that might apply to the valve; 
   // similarly, the PERMISSIVE, INTERLOCK and TRIP parameters are the links to any such interlock 
   // signals that may be applied to the device.
   // 
   // The STATIC_DATA and DYNAMIC_DATA parameters are UDTs that hold (respectively) the 
   // configuration information and the live data for the device.
   // 
   //  ――――――――――――――――――――――――――――――――――――――――――
   //  PARAM         ASSOCIATED UDT          ASSOCIATED DATA BLOCK
   //  ――――――――――――――――――――――――――――――――――――――――――
   //  STATIC_DATA     UT11101_St_DevValveBi           DB11101_St_DevValveBi
   //  DYNAMIC_DATA   UT31101_Dy_DevValveBi           DB31101_Dy_DevValveBi
   //  ――――――――――――――――――――――――――――――――――――――――――
   // 
   // 
   // Section 6 contains a full list of all variables within these UDTs.
   // 
   // This arrangement conforms with the PAL philosophy where IO card connections, safety 
   // signals and interlocks have unique formal parameters; all remaining signals are passed as 
   // variables within UDTs, see the Software Design Specification [Ref. 008].
   // 
   // 
   // 
   // ▂▂▂▂▂▂▂▂▂▂▂▂▂▂▂▂▂▂▂▂▂▂▂▂▂▂▂▂▂▂▂▂▂▂▂▂▂▂▂▂▂▂▂▂
   // 3.1      Typical wiring arrangement
   // 
   // 
   // The typical wiring arrangements for a valve with all signals is as follows:
   // 
   //     24VDC  
   //      ─┬─                                ┌──────┬───┐
   //       │                                 │         │   │
   //       ├────┬────┐                 │         │  ─┴─
   //       │       │       │                 │         │    GND
   //       │       │       │             ┌┻┐ ▁▁ ┌┻┐
   //    ▁│ ○   ▁│○   ▁│○             │ │▁＼／▁│ │
   //    ▔│ ○   ▔│○   ▔│○             │ │ ／＼ │ │
   //     FAULT│ CLOSED│   OPEN│             └┬┘ ▔▔ └┬┘
   //       │       │       │                 │         │
   //       │       │       │              │         │
   //     ┌─┻─┐┌─┻─┐┌─┻─┐          ┌─┻─┐  ┌─┻─┐
   //     │  I1.0  ││  I1.1  ││  I1.2  │DI CARD        │  Q1.0 │  │  Q1.1 │DO CARD
   //     └─┬─┘└─┬─┘└─┬─┘          └─┬─┘  └─┬─┘
   //       │       │       │ ┌────────    │      │
   //       │       │       │ │ FC11101          │      │
   //       │       │       │ ├──────────┤ │      │
   //       │       │       │ │          │ │      │
   //       │       │       │ │          OPEN_CMD ├─┘      │
   //       │       │       │ │          │        │
   //       │       │       │ │     CLOSE_CMD ├────────┘
   //       │       │       │ │          │
   //       │       │       └─┤ FBK_OPEN        │
   //       │       │         │          │
   //       │       └──────┤ FBK_CLOSED       │
   //       │                 │          │
   //       └───────────┤ EXT_FAULT        │
   //                         │
   //                         │
   // 
   // 
   // 
   // ▂▂▂▂▂▂▂▂▂▂▂▂▂▂▂▂▂▂▂▂▂▂▂▂▂▂▂▂▂▂▂▂▂▂▂▂▂▂▂▂▂▂▂▂
   // 3.2      Normal operation 
   // 
   // 
   // Normal operation can generally be considered the operation of both normally open and normally 
   // closed valves under automatic or manual control (see § 3.5.1 for a full explanation of how 
   // automatic and manual modes are selected). And the mechanisms used to determine the state 
   // of the valve.
   // 
   // 
   // 
   // ▁▁▁▁▁▁▁▁▁▁▁▁▁▁▁▁▁▁▁▁▁▁▁▁▁▁▁▁▁▁▁▁▁▁▁▁▁▁▁▁▁▁▁▁
   // 3.2.1     Opening and closing the valve
   // 
   // 
   // Under automatic mode, the valve is controlled by separate software within the Controller (this 
   // is usually derived from either continuous control logic or sequential control logic and 
   // implemented by the command handling application module).
   // 
   // The result of this software will be to either open the valve or close the valve.
   // 
   // Under manual mode, the valve is controlled directly by the operator via some form of 
   // supervisory system (SCADA or HMI). Again, the result of the manual operator action will be to 
   // either open or close the valve.
   // 
   // There are two signals that, under normal operation, can cause the valve to move to a particular 
   // state, one for automatic mode and one for manual mode, both are passed to the module as 
   // part of the DYNAMIC_DATA parameter (UT31101_Dy_DevValveBi):
   // 
   // 
   //  DATA STRUCTURE    UT31101_Dy_DevValveBi
   //  ――――――――――――――――――――――――――――――――――――――――――
   //  SIGNAL         FUNCTION               TYPE     DETAILS
   //  ――――――――――――――――――――――――――――――――――――――――――
   //  ctrl_Aut_OpenClose Causes the valve to open and close     Bool  1 = open the valve
   //            if automatic mode is active            0 = close the valve
   //            (mode_AutMan = 1). If auto mode is 
   //            not active, signal is ignored
   // 
   //  ctrl_Man_OpenClose  Causes the valve to open and close     Bool  1 = open the valve
   //            if manual mode is active             0 = close the valve
   //            (mode_AutMan = 0). If man mode is 
   //            not active, signal is ignored
   //  ――――――――――――――――――――――――――――――――――――――――――
   // 
   // The operating mode (either automatic or manual) is specified within the DYNAMIC_DATA 
   // parameter UDT (UT31101_Dy_DevValveBi) mode_AutMan as follows:
   // 
   // 
   //  DATA STRUCTURE    UT31101_Dy_DevValveBi
   //  ――――――――――――――――――――――――――――――――――――――――――
   //  SIGNAL         FUNCTION               TYPE     DETAILS
   //  ――――――――――――――――――――――――――――――――――――――――――
   //  Mode_AutMan     Identifies the operating mode of     Bool  1 = automatic mode
   //            the valve.                   0 = manual mode
   //  ――――――――――――――――――――――――――――――――――――――――――
   // 
   // It is possible to configure the module such that manual mode is permanently disabled; this uses 
   // the following STATIC_DATA parameter:
   // 
   //  DATA STRUCTURE    UT11101_St_DevValveBi
   //  ――――――――――――――――――――――――――――――――――――――――――
   //  SIGNAL         FUNCTION               TYPE     DETAILS
   //  ――――――――――――――――――――――――――――――――――――――――――
   //  CONFIG_MAN_DIS     Prevents manual mode being       Bool  1 = no manual mode
   //            activated under all circumstances            0 = manual permitted
   //            device is in auto, Mode_AutMan is 
   //            set permanently to 1
   //  ――――――――――――――――――――――――――――――――――――――――――
   // 
   // If manual mode is disabled (configuration signal CONFIG_MAN_DIS is set to 1), then manual 
   // mode cannot be turned on under any circumstances, the option will be greyed out on the 
   // supervisory system faceplate and the module will constantly set the mode_AutMan signal to 1.
   // 
   // By default the device will be in automatic mode.
   // 
   // The state of the OPEN_CMD and CLOSE_CMD parameters is determined by either the 
   // ctrl_Aut_OpenClose or ctrl_Man_OpenClose (depending on whether automatic mode or 
   // manual mode is active) and whether the outputs are configured to deenergise or remain active 
   // (maintained) when the valve reaches the desired state.
   // 
   // The facility to deenergise outputs or for them to be maintained once the required state is reached 
   // is determined using the following STATIC_DATA parameter:
   // 
   // 
   //  DATA STRUCTURE    UT11101_St_DevValveBi
   //  ――――――――――――――――――――――――――――――――――――――――――
   //  SIGNAL         FUNCTION               TYPE     DETAILS
   //  ――――――――――――――――――――――――――――――――――――――――――
   //  CONFIG_MAINT_OP    If set to 1, either the OPEN _CMD or   Bool  1 = Maintain outputs
   //            CLOSE_CMD will remain active when       0 = deenergise output
   //            the valve reaches the required state.
   // 
   //            If set to 0, the OPEN _CMD and  
   //            CLOSE_CMD will deenergise after the 
   //            run-on timer is complete.
   //  ――――――――――――――――――――――――――――――――――――――――――
   // 
   // The various states of the valve for both automatic and manual operations are given in the following 
   // tables. The first table shows the output states for deenergising outputs, the second for maintained 
   // outputs:
   // 
   // 
   //  ――――――――――――――――――――――――――――――――――――――――――
   //  MODE:   AUTOMATIC MODE (mode_AutMan = 1)
   //      and outputs configured to deenergise (CONFIG_MAINT_OP = 0)
   // 
   //  ctrl_Aut_OpenClose ctrl_Man_OpenClose OPEN_CMD      CLOSE_CMD  VALVE STATE
   //  ――――――――――――――――――――――――――――――――――――――――――
   //      0         N/A      0         1          Closing
   //      1         N/A      1         0          Opening
   //      0         N/A      0         0          Closed
   //      1         N/A      0         0          Open
   //  ――――――――――――――――――――――――――――――――――――――――――
   // 
   //  MODE:   MANUAL MODE (mode_AutMan = 0)
   //      and outputs configured to deenergise (CONFIG_MAINT_OP = 0)
   // 
   //  ctrl_Aut_OpenClose ctrl_Man_OpenClose OPEN_CMD      CLOSE_CMD  VALVE STATE
   //  ――――――――――――――――――――――――――――――――――――――――――
   //       N/A          0       0         1          Closing
   //       N/A          1       1         0          Opening
   //       N/A          0       0         0          Closed
   //       N/A          1       0         0          Open
   //  ――――――――――――――――――――――――――――――――――――――――――
   //    Once the valve has reached its requested state (open or closed), the OPEN_CMD and 
   //    CLOSE_CMD outputs are deenergised after the run-on timer is complete
   // 
   // 
   //  ――――――――――――――――――――――――――――――――――――――――――
   //  MODE:   AUTOMATIC MODE (mode_AutMan = 1)
   //      and outputs configured to be maintained  (CONFIG_MAINT_OP = 1)
   // 
   //  ctrl_Aut_OpenClose ctrl_Man_OpenClose OPEN_CMD      CLOSE_CMD  VALVE STATE
   //  ――――――――――――――――――――――――――――――――――――――――――
   //      0         N/A      0         1          Closing
   //      1         N/A      1         0          Opening
   //      0         N/A      0         0          Closed
   //      1         N/A      0         0          Open
   //  ――――――――――――――――――――――――――――――――――――――――――
   // 
   //  MODE:   MANUAL MODE (mode_AutMan = 0)
   //      and outputs configured to be maintained  (CONFIG_MAINT_OP = 1)
   // 
   //  ctrl_Aut_OpenClose ctrl_Man_OpenClose OPEN_CMD      CLOSE_CMD  VALVE STATE
   //  ――――――――――――――――――――――――――――――――――――――――――
   //       N/A          0       0         1          Closing
   //       N/A          1       1         0          Opening
   //       N/A          0       0         0          Closed
   //       N/A          1       1         1          Open
   //  ――――――――――――――――――――――――――――――――――――――――――
   //    Once the valve has reached its requested state (open or closed), the OPEN_CMD and 
   //    CLOSE_CMD outputs remain active
   // 
   // If the valve is in a fault state (see § 3.3), both the OPEN_CMD and CLOSE_CMD parameters will be 
   // set to 0 (deenergised), irrespective of any other signals.
   // 
   // 
   // 
   // ▁▁▁▁▁▁▁▁▁▁▁▁▁▁▁▁▁▁▁▁▁▁▁▁▁▁▁▁▁▁▁▁▁▁▁▁▁▁▁▁▁▁▁▁
   // 3.2.2     A note on maintained output signals
   // 
   // 
   // A bistable valve is usually configured to either deenergise the OPEN_CMD and CLOSE_CMD 
   // output signals when the valve reaches its demanded position (after a specified run-on time), 
   // it can also be configured to permanently maintain the ap-propriate output the signal when the 
   // demanded position is reached.
   // 
   // The default arrangement is for the output signals to automatically deenergise once the valve 
   // reaches position (bistable valves generally only require the driving signals to be applied when 
   // the valve is changing state). 
   // 
   // The maintain option is selected by setting CONFIG_MAINT_OP to a value of 1, deenergise mode 
   // is selected by setting CONFIG_MAINT_OP to a value of 0.
   // 
   // The option to maintain the outputs when the demanded state is reached, although not normally 
   // required, is provided and may be used if deemed necessary.
   // 
   // Note:    If the option to maintain the outputs is activated, the valve must be rated to have its 
   //      actuating signals permanently energised.
   // 
   // If the maintain option is active, the outputs will still deenergise if a fault is detected.
   // 
   // 
   // 
   // ▁▁▁▁▁▁▁▁▁▁▁▁▁▁▁▁▁▁▁▁▁▁▁▁▁▁▁▁▁▁▁▁▁▁▁▁▁▁▁▁▁▁▁▁
   // 3.2.3     Operation timers
   // 
   // 
   // The module an operation timer used for both opening the valve and for closing the valve.
   // 
   // The timer is loaded with either the opening operation time or closing operation time whenever 
   // the valve is requested to change state. The timer counts down from the loaded value to zero 
   // (the valve can have different times for opening and closing).
   // 
   // The specific operating times are given within the STATIC_DATA parameter 
   // UDT (UT11101_St_DevValveBi) as follows:
   // 
   // 
   //  DATA STRUCTURE    UT11101_St_DevValveBi
   //  ――――――――――――――――――――――――――――――――――――――――――
   //  SIGNAL         FUNCTION               TYPE     DETAILS
   //  ――――――――――――――――――――――――――――――――――――――――――
   //  TIME_OPENING_MAX The maximum time required for the     Real     Time in seconds
   //            valve to travel from a closed state to
   //            an open state
   // 
   //  TIME_CLOSING_MAX The maximum time required for the     Real     Time in seconds
   //            valve to travel from an open state to 
   //            a closed state
   //  ――――――――――――――――――――――――――――――――――――――――――
   // 
   // If the timer is running, the elapsed (counting down) time is stored within the DYNAMIC_DATA 
   // parameter UDT (UT31101_Dy_DevValveBi) as follows:
   // 
   // 
   //  DATA STRUCTURE    UT31101_Dy_DevValveBi
   //  ――――――――――――――――――――――――――――――――――――――――――
   //  SIGNAL           FUNCTION               TYPE     DETAILS
   //  ――――――――――――――――――――――――――――――――――――――――――
   //  actual_Operating_Timer    The actual elapsed operation time       Real     Time in seconds
   //  ――――――――――――――――――――――――――――――――――――――――――
   // 
   // There is a single operating timer for both opening and closing (opening and closing are mutually 
   // exclusive operations, hence only one timer is needed. The timer is preloaded with either the 
   // opening time preset or the closing time preset prior to the timer starting).
   // 
   // The preset signals TIME_OPENING_MAX and TIME_CLOSING_MAX are the maximum possible 
   // times it can take for the valve to reach the expected position. This should be set to between 
   // 110% and 120% of the normal opening and closing times specified for the valve. For example, 
   // if a valve has a normal opening time of 5 seconds and a normal closing time of 3 seconds, 
   // sensible values for TIME_OPENING_MAX and TIME_CLOSING_MAX would be between 5.5-6.0 s 
   // and 3.3-4.0 s respectively.
   // 
   // A valve will enter a fault state (see § 3.4) if the operation timer counts down to a value of zero 
   // without confirmation that the valve has reached the required state. Such confirmation is 
   // provided by positive feedback from the valve limit switches (or other indicating devices) or 
   // by simulated signal within the module itself (see § 3.2.3).
   // 
   // The operation timer always counts down from a preset value to zero, this is in accordance 
   // with the general requirements and practices of the PAL software.
   // 
   // 
   // 
   // ▁▁▁▁▁▁▁▁▁▁▁▁▁▁▁▁▁▁▁▁▁▁▁▁▁▁▁▁▁▁▁▁▁▁▁▁▁▁▁▁▁▁▁▁
   // 3.2.4     Run-on timers
   // 
   // 
   // The module has a run-on timer that activates whenever a valve that is changing state, reaches 
   // the demanded position. The run-on timer is used to maintain either the OPEN_CMD or 
   // CLOSE_CMD output for a short time period after the valve has reached the demanded position 
   // to ensure that the valve is firmly in position (it pre-vents the valve stopping the instant the limit 
   // switch confirms the valve position, it provides some hysteresis to ensure that the valve is 
   // positively in position before deactivating the driving signals).
   // 
   // Different values can be specified for the run-on timer, depending whether the valve is opening 
   // or closing.
   // 
   // The run-on timer is loaded with either the opening run-on time or closing run-on time 
   // whenever the valve is requested to change state. The timer begins to count down from the 
   // loaded value to zero, the instant the valve reaches position (and the operation timer stops). The 
   // valve can have different run-on times for opening and closing.
   // 
   // The specific run-on times are given within the STATIC_DATA parameter UDT 
   // (UT11101_St_DevValveBi) as follows:
   // 
   // 
   //  DATA STRUCTURE    UT11101_St_DevValveBi
   //  ――――――――――――――――――――――――――――――――――――――――――
   //  SIGNAL           FUNCTION               TYPE DETAILS
   //  ――――――――――――――――――――――――――――――――――――――――――
   //  TIME_OPENING_RUNON    The run-on time period activated when     Real  Time in seconds
   //              the valve reaches the open position
   //              OPEN_CMD will be maintained for this 
   //              period
   // 
   //  TIME_CLOSING_RUNON    The run-on time period activated when     Real  Time in seconds
   //              the valve reaches the closed position
   //              CLOSE_CMD will be maintained for this 
   //              period
   //  ――――――――――――――――――――――――――――――――――――――――――
   // 
   // If the run-on timer is active, the elapsed (counting down) time is stored within the DYNAMIC_DATA 
   // parameter UDT (UT31101_Dy_DevValveBi) as follows:
   // 
   // 
   //  DATA STRUCTURE    UT31101_Dy_DevValveBi
   //  ――――――――――――――――――――――――――――――――――――――――――
   //  SIGNAL           FUNCTION               TYPE DETAILS
   //  ――――――――――――――――――――――――――――――――――――――――――
   //  actual_Runon_Timer     Actual (elapsed) value of the run-on timer   Real  Time in seconds
   //  ――――――――――――――――――――――――――――――――――――――――――
   // 
   // There is a single run-on timer for both the opening and closing run-on operations (opening and 
   // closing are mutually exclusive operations, hence only one timer is needed. The timer is 
   // preloaded with either the opening run-on time preset or the closing run-on time preset prior to 
   // the timer starting).
   // 
   // The effect of the run-on timer is shown graphically below: 
   // 
   // 
   // │   ┌────────────────┐
   // │   │                │
   // │   │                │            ctrl_Aut_OpenClose
   // │   │                │
   // ┼───┘┈┈┈┈┈┈┈┈┈┈┈┈┈┈┈┈└───────────────
   //     ╎                ╎
   //     ╎                ╎
   // │   ╎      ┌──────────┐
   // │   ╎      │         ╎│
   // │   ╎      │         ╎│             FBK_OPEN
   // │   ╎      │         ╎│
   // ┼──────────┘┈┈┈┈┈┈┈┈┈┈└────────────────
   //     ╎
   // │────┐     ╎         ╎       ┌───────
   // │   ╎│     ╎         ╎       │
   // │   ╎│     ╎         ╎       │               FBK_CLOSED
   // │   ╎│     ╎         ╎       │
   // ┼┈┈┈┈└───────────────────────┘┈┈┈┈┈┈┈
   //     ╎      ╎         ╎       ╎
   //     ↓            ↓                  ↓       ↓          
   // │   ┌──────┐         ┌───────┐   
   // │   │      │         │       │  
   // │   │←    Ａ  →│         │←      Ｂ    →│  actual_Operating_Timer
   // │   │      │         │       │  
   // ┼───┘┈┈┈┈┈┈└─────────┘┈┈┈┈┈┈┈└───────
   //     ╎      ╎         ╎       ╎
   //     ╎      ↓         ╎       ↓
   // │   ╎      ┌──┐      ╎       ┌─┐   
   // │   ╎      │  Ｃ  │      ╎       │Ｄ│  
   // │   ╎      │  │      ╎       │ │    actual_Runon_Timer
   // │   ╎      │  │      ╎       │ │  
   // ┼──────────┘┈┈└──────────────┘┈└───────
   //     ╎         ╎      ╎         ╎
   //     ↓               ↓      ╎         ╎         
   // │   ┌─────────┐      ╎         ╎   
   // │   │         │      ╎         ╎  
   // │   │         │      ╎         ╎    OPEN_CMD
   // │   │         │      ╎         ╎  
   // ┼───┘┈┈┈┈┈┈┈┈┈└────────────────────────
   // 
   //                      ╎         ╎
   //                      ↓               ↓ 
   // │                    ┌─────────┐  
   // │                    ╎         ╎  
   // │                    ╎         ╎    CLOSE_CMD
   // │                    ╎         ╎  
   // ┼────────────────────┘┈┈┈┈┈┈┈┈┈└───────
   // 
   // 
   //   Ａ Operation timer (opening)
   //   Ｂ Operation timer (closing)
   //   Ｃ Run-on timer (opening)
   //   Ｄ Run-on timer (closing)
   // 
   // The run-on timer starts on the falling edge of the operation timer (this in turn is determined by 
   // the valve reaching the correct position).
   // 
   // The preset signals TIME_OPENING_RUNON and TIME_CLOSING_RUNON cause the OPEN_CMD and 
   // CLOSE_CMD signals (respectively) to remain active for a period after the appropriate limit switch 
   // positions have been reached
   // 
   // The run-on timer always counts down from a preset value to zero, this is in accordance with the 
   // general requirements and practices of the PAL software.
   // 
   // If the valve is required to change state while the run-on timer is active, the run-on timer will 
   // simply stop (effectively be cancelled) until required to run again at the end of the operation timer.
   // 
   // If the valve is in a fault condition (i.e. if the valve did not achieve the correct state), the run-on 
   // timer will not activate.
   // 
   // The recovery timer will always run after a fault condition is reset (even an external fault), this 
   // ensures that the valve movement operation is fully completed.
   // 
   // The run-on timer will not activate under any circumstances if the module is configured to 
   // maintain its outputs (CONFIG_MAINT_OP = 1).
   // 
   // 
   // 
   // ▁▁▁▁▁▁▁▁▁▁▁▁▁▁▁▁▁▁▁▁▁▁▁▁▁▁▁▁▁▁▁▁▁▁▁▁▁▁▁▁▁▁▁▁
   // 3.2.5     Operation with maintained outputs
   // 
   // If the module is configured to maintain the OPEN_CMD and CLOSE_CMD signals when the 
   // required state is reached (CONFIG_MAINT_OP = 1), the run-on timer will not activate under any 
   // circumstances and the operation diagram becomes:
   // 
   // 
   // 
   // 
   // │   ┌────────────────┐
   // │   │                │
   // │   │                │            ctrl_Aut_OpenClose
   // │   │                │
   // ┼───┘┈┈┈┈┈┈┈┈┈┈┈┈┈┈┈┈└───────────────
   //     ╎                ╎
   //     ╎                ╎
   // │   ╎      ┌──────────┐
   // │   ╎      │         ╎│
   // │   ╎      │         ╎│             FBK_OPEN
   // │   ╎      │         ╎│
   // ┼──────────┘┈┈┈┈┈┈┈┈┈┈└────────────────
   //     ╎
   // │────┐     ╎         ╎       ┌───────
   // │   ╎│     ╎         ╎       │
   // │   ╎│     ╎         ╎       │               FBK_CLOSED
   // │   ╎│     ╎         ╎       │
   // ┼┈┈┈┈└───────────────────────┘┈┈┈┈┈┈┈
   //     ╎      ╎         ╎       ╎
   //     ↓            ↓                  ↓       ↓          
   // │   ┌──────┐         ┌───────┐   
   // │   │      │         │       │  
   // │   │←    Ａ  →│         │←      Ｂ    →│  actual_Operating_Timer
   // │   │      │         │       │  
   // ┼───┘┈┈┈┈┈┈└─────────┘┈┈┈┈┈┈┈└───────
   //     ╎                ╎          
   //     ↓                      ↓                   
   // │   ┌────────────────┐                    
   // │   │                │                   
   // │   │                │              OPEN_CMD
   // │   │                │                   
   // ┼───┘┈┈┈┈┈┈┈┈┈┈┈┈┈┈┈┈└─────────────────
   //     ╎                ╎
   //     ↓                      ↓
   // │───┐                ┌─────────────────  
   // │   ╎                ╎            
   // │   ╎                ╎              CLOSE_CMD
   // │   ╎                ╎            
   // ┼┈┈┈└────────────────┘┈┈┈┈┈┈┈┈┈┈┈┈┈┈┈┈┈
   // 
   // 
   //   Ａ Operation timer (opening)
   //   Ｂ Operation timer (closing)
END_REGION

REGION Network 3: Block description — Section 3.2.6 to 3.2.8
   // ▁▁▁▁▁▁▁▁▁▁▁▁▁▁▁▁▁▁▁▁▁▁▁▁▁▁▁▁▁▁▁▁▁▁▁▁▁▁▁▁▁▁▁▁
   // 3.2.6     Position feedback signals
   // 
   // 
   // The module can accommodate either none, one or two positive position indication signals:
   // 
   // 
   //    1.  No limit switches         There is no positive indication of the current state 
   //                      of the valve, it is assumed to be in the expected 
   //                      state.
   // 
   //    2.  Closed limit switch only       Positive indication is given for the closed state 
   //                      only. The valve is assumed to be open if the 
   //                      closed signal is inactive.
   // 
   //    3.  Open limit switch only      Positive indication is given for the open state 
   //                      only. The valve is assumed to be closed if the 
   //                      open signal is inactive.
   // 
   //    4.  Open and closed limit switches    Positive indication is given for both states. 
   //                      This allows the true state of the valve to be 
   //                      determined under all circumstances.
   // 
   // There are two configuration signals that determine the position feedback arrangements, these 
   // are stored within the STATIC_DATA parameter UDT as follows:
   // 
   // 
   //  DATA STRUCTURE    UT11101_St_DevValveBi
   //  ――――――――――――――――――――――――――――――――――――――――――
   //  SIGNAL           FUNCTION              TYPE     DETAILS
   //  ――――――――――――――――――――――――――――――――――――――――――
   //  CONFIG_FBK_OPEN_EN    Indicates that positive feedback for    Bool  1 = open feedback
   //              the open state is present           0 = no feedback
   // 
   //  CONFIG_FBK_CLOSED_EN  Indicates that positive feedback for    Bool  1 = closed feedback
   //              the closed state is present            0 = no feedback
   //  ――――――――――――――――――――――――――――――――――――――――――
   // 
   // If the CONFIG_FBK_OPEN_EN signal is activated (set to 1), the module will use the state of the 
   // signal connected to the FBK_OPEN parameter to determine the open position of the valve. 
   // 
   // If the CONFIG_FBK_OPEN_EN signal is deactivated (set to 0), the module will derive the open 
   // position of the valve such that it matches the requested state of the valve.
   // 
   // Similarly, if the CONFIG_FBK_CLOSED_EN signal is activated (set to 1), the module will use the 
   // state of the signal connected to the FBK_CLOSED parameter to determine the closed position of 
   // the valve. 
   // 
   // If the CONFIG_FBK_CLOSED_EN signal is deactivated (set to 0), the module will derive the 
   // closed position of the valve such that it matches the requested state of the valve.
   // 
   // Where a CONFIG_FBK_OPEN/CLOSED_EN signal is activated (set to 1), a true state on the 
   // associated parameter FBK_OPEN/CLOSED indicates that the valve is in that position, a false 
   // state indicates that the valve is not in that position as follows:
   // 
   //  OPEN SIGNALS  ―――――――――――――――――――――――――――――――――――
   //  CONFIG_FBK_OPEN_EN    FBK_OPEN    MEANING
   //  ――――――――――――――――――――――――――――――――――――――――――
   //       1            0       Not open
   //       1            1       Confirmed open
   //       0          N/A     Internally derived open signal matches
   //                        requested valve state, FBK_OPEN is ignored
   //  ――――――――――――――――――――――――――――――――――――――――――
   // 
   // 
   //  CLOSED SIGNALS ――――――――――――――――――――――――――――――――――
   //  CONFIG_FBK_CLOSED_EN  FBK_CLOSED  MEANING
   //  ――――――――――――――――――――――――――――――――――――――――――
   //       1            0       Not closed
   //       1            1       Confirmed closed
   //       0          N/A     Internally derived closed signal matches
   //                        requested valve state, FBK_CLOSED is ignored
   //  ――――――――――――――――――――――――――――――――――――――――――   
   // 
   // 
   // 
   // 
   // ▁▁▁▁▁▁▁▁▁▁▁▁▁▁▁▁▁▁▁▁▁▁▁▁▁▁▁▁▁▁▁▁▁▁▁▁▁▁▁▁▁▁▁▁
   // Position status signals
   // 
   // 
   // The true position of the valve is given as status signals:
   // 
   //  DATA STRUCTURE    UT31101_Dy_DevValveBi
   //  ――――――――――――――――――――――――――――――――――――――――――
   //  SIGNAL          FUNCTION                TYPE     DETAILS
   //  ――――――――――――――――――――――――――――――――――――――――――
   //  status_Closed      Valve is confirmed closed         Bool     1 = closed
   //                                    0 = not closed
   // 
   //  status_Opening      Valve is opening             Bool     1 = opening
   //                                    0 = not opening
   // 
   //  status_Open      Valve is confirmed open         Bool     1 = open
   //                                    0 = not open
   // 
   //  status_Closing     Valve is closing               Bool     1 = closing
   //                                    0 = not closing
   // 
   //  status_Operating      Valve is changing state          Bool     1 = changing state
   //             (either opening or closing)           0 = fixed state
   // 
   //  status_Fault       Valve is in a fault condition          Bool     1 = fault
   //                                    0 = healthy
   //  ――――――――――――――――――――――――――――――――――――――――――   
   // 
   // The standard arrangement is for symbols to show discrete opening and closing symbols; there 
   // are some instances (usually on less sophisticated HMIs) where it is necessary to show only that 
   // the valve is in the process of changing state.
   // 
   // This is achieved through the use of the status_Operating signal (this is active whenever either 
   // status_Opening or status_Closing is active), status_Operating indicates that the valve is either 
   // opening or closing, but does not distinguish which.
   // 
   // 
   // 
   // ▁▁▁▁▁▁▁▁▁▁▁▁▁▁▁▁▁▁▁▁▁▁▁▁▁▁▁▁▁▁▁▁▁▁▁▁▁▁▁▁▁▁▁▁
   // Understanding derived position signals
   // 
   // 
   // Where either the CONFIG_FBK_OPEN_EN or CONFIG_FBK_CLOSED_EN signal is deactivated 
   // (set to 0), the associated position feedback is internally determined by the module according to 
   // the actual state of the valve (determined by the OPERATE parameter and the type of valve in use).
   // 
   // These internally derived signals are themselves configurable and can be set such that the 
   // position feedback signal occurs after a particular percentage of the associated operation timer 
   // has expired.
   // 
   // For the derived FBK_OPEN signal, the configurable percentage signal is TIME_DER_OPEN 
   // stored within the STATIC_DATA parameter. Similarly, for the derived FBK_CLOSED signal, the 
   // configurable percentage signal is TIME_DER_CLOSED, again, stored within the STATIC_DATA 
   // parameter.
   // 
   // The operation of these parameters can be seen below:
   // 
   //     ①                ③
   // │   ┌────────────────┐
   // │   │                │
   // │   │                │      ctrl_Aut_OpenClose
   // │   │                │
   // ┼───┘┈┈┈┈┈┈┈┈┈┈┈┈┈┈┈┈└───────────────
   // 
   // 
   //                      TIME_OPENING_MAX            TIME_CLOSING_MAX
   //      ←         →       ←                →
   // │   ┌──────┐┄┄┐      ┌───────┐┄┄┐
   // │   │      │  ┆      │       │  ┆
   // │   │←    Ａ  →│  ┆      │←      Ｂ    →│  ┆actual_Operating_Timer
   // │   │      │  ┆      │       │  ┆
   // ┼───┘┈┈┈┈┈┈└──┴──────┘┈┈┈┈┈┈┈└──┴────
   //     ╎      ②         ╎       ④
   //     ╎      ╎         ╎       ╎
   //     ↓      ╎         ╎       ↓
   // │───┐      ╎         ╎       ┌───────
   // │   │      ╎         ╎       │
   // │   │      ╎         ╎       │                FBK_CLOSED (derived)
   // │   │      ╎         ╎       │
   // ┼┈┈┈└────────────────────────┘┈┈┈┈┈┈┈
   //     Ｃ      ╎         ╎       Ｆ
   //            ╎         ╎
   //            ╎         ╎
   //            ↓         ↓
   // │          ┌─────────┐
   // │          │         │
   // │          │         │               FBK_OPEN (derived)
   // │          │         │
   // ┼──────────┘┈┈┈┈┈┈┈┈┈└────────────────
   //            Ｄ         Ｅ
   // 
   //   Ａ TIME_DER_OPEN  (95%)
   //   Ｂ TIME_DER_CLOSED  (80%)
   //   Ｃ Closed signal deactivates instantly when the valve is asked to open
   //   Ｄ Open signal activates when actual_Operating_Timer reaches TIME_DER_OPEN 
   //     as a percentage of TIME_OPENING_MAX
   //   Ｅ Open signal deactivates instantly when the valve is asked to close
   //   Ｆ Closed signal activates when actual_Operating_Timer reaches TIME_DER_CLOSED 
   //     as a percentage of TIME_CLOSING_MAX
   // 
   // The figure above assumes a normally closed valve with no position feedback signals (both 
   // CONFIG_FBK_OPEN_EN and CONFIG_FBK_CLOSED_EN are set to 0) operating in automatic mode. 
   // It also assumes that the valve is free to operate without restriction (there are no active interlock 
   // or safety signals).
   // 
   // The valve is initially closed with the derived FBK_CLOSED signal active (1) and the derived 
   // FBK_OPEN signal deactivated (0). At some point 1, the module receives a request to open the 
   // valve.
   // 
   // At this point two things happen, firstly the operation timer starts, with a countdown from the 
   // value TIME_OPENING_MAX, which in this case is 3 seconds. Secondly, the derived FBK_CLOSED 
   // signal is deenergised (indicating the valve is no longer closed).
   // 
   // The simulated opening time (TIME_DER_OPEN) is set to 95%, this means that the derived 
   // FBK_OPEN signal will activate when the actual_Operating_Timer value has counted down for 
   // 95% of the TIME_OPENING_MAX value (i.e. when the timer has counted down to 0.15s or less). 
   // 
   // The exact formula used is:
   // 
   // ┌───────────────────────────────────────────┐
   // │Derived FBK_OPEN=1 when:                                     │
   // │                                 TIME_DER_OPEN        │
   // │actual_Operating_Timer ≤ TIME_OPENING_MAX ─ TIME_OPENING_MAX ╳ --------------------------------        │
   // │                                     100     │
   // └───────────────────────────────────────────┘
   // 
   // This can be seen at point ②, where the derived FBK_OPEN signal activates. The valve now 
   // remains in the open state (FBK_OPEN = 1. FBK_CLOSED = 0) until there is a request to close 
   // the valve, point ③.
   // 
   // Again, at point ③, the module receives a request to close the valve.
   // 
   // At this point two things happen, firstly the operation timer starts, with a countdown from the 
   // value TIME_CLOSING_MAX, which in this case is 4 seconds. Secondly, the derived FBK_OPEN signal 
   // is deenergised (indicating the valve is no longer open).
   // 
   // The simulated closing time (TIME_DER_CLOSED) is set to 80%, this means that the derived 
   // FBK_CLOSED signal will activate when the actual_Operating_Timer value has counted down 
   // for 80% of the TIME_CLOSING_MAX value (i.e. when the timer has counted down to 0.80s or less). 
   // 
   // The exact formula used is:
   // 
   // ┌────────────────────────────────────────────┐
   // │Derived FBK_CLOSED=1 when:                               │
   // │                                 TIME_DER_CLOSED          │
   // │actual_Operating_Timer ≤ TIME_CLOSING_MAX ─ TIME_CLOSING_MAX ╳ ------------------------------------         │
   // │                                     100            │
   // └────────────────────────────────────────────┘
   // 
   // This can be seen at point ④, where the derived FBK_CLOSED signal activates. The valve now 
   // remains in the closed state (FBK_OPEN = 0. FBK_CLOSED = 1) until there is a request a 
   // subsequent request to reopen the valve.
   // 
   // If only one position feedback is derived (the other being an actual signal), then the derived signal 
   // will be generated in exactly the same way as above, the non-derived signal will simply use the 
   // true status of the signal passed as a parameter to the module.
   // 
   // The simulated time signals are passed to the module within the STATIC_DATA parameter 
   // UDT (UT11101_St_DevValveBi) as follows:
   // 
   //  DATA STRUCTURE    UT11101_St_DevValveBi
   //  ――――――――――――――――――――――――――――――――――――――――――
   //  SIGNAL        FUNCTION              TYPE     DETAILS
   //  ――――――――――――――――――――――――――――――――――――――――――
   //  TIME_DER_CLOSED           Specifies the percentage of the     Real     Percentage
   //              TIME_OPENING_MAX value that 
   //              must expire before the derived 
   //              FBK_OPEN signal activates.
   // 
   // 
   //  TIME_DER_OPEN             Specifies the percentage of the     Real     Percentage
   //              TIME_CLOSING_MAX value that 
   //              must expire before the derived 
   //              FBK_CLOSED signal activates.
   //  ――――――――――――――――――――――――――――――――――――――――――
   // 
   // Both configuration signals are restricted to the range 0.00-100.00, the default value is 90% for 
   // both open and closed.
   // 
   // 
   // 
   // ▁▁▁▁▁▁▁▁▁▁▁▁▁▁▁▁▁▁▁▁▁▁▁▁▁▁▁▁▁▁▁▁▁▁▁▁▁▁▁▁▁▁▁▁
   // 3.2.7    Recording the last operation time
   // 
   // 
   // The module records the last complete operation time value, it records the actual time taken for 
   // the valve to reach the correct designated position.
   // 
   // For example if the valve received a request to open, and it required 4.8 seconds for the position 
   // feedback to report the correct (open) state, the module would record a value of 4.8 seconds in 
   // the actual_Last_Op_Time value (passed as part of the DYNAMIC_DATA parameter).
   // 
   // Similarly, if the valve were requested to close, and required 6.2 seconds for the position feedback 
   // to report the correct (closed) state, the module would record a value of 6.2 seconds in the 
   // actual_Last_Op_Time value.
   // 
   // The actual_Last_Op_time value forms part of the DYNAMIC_DATA parameter UDT as follows:
   // 
   // 
   //  DATA STRUCTURE    UT31101_Dy_DevValveBi
   //  ――――――――――――――――――――――――――――――――――――――――――
   //  SIGNAL        FUNCTION              TYPE     DETAILS
   //  ――――――――――――――――――――――――――――――――――――――――――
   //  actual_Last_Op_Time     Stores the actual time taken for     Real     Time in seconds
   //             the valve to achieve the correct 
   //             open or closed state.
   // 
   //             Receives a value of -1.0 if the 
   //             valve did not achieve the correct 
   //             position in the specified 
   //             operation time
   //  ――――――――――――――――――――――――――――――――――――――――――
   // 
   // If the valve does not achieve the requested position (within either the TIME_OPENING_MAX or 
   // TIME_CLOSING_MAX limits), a value of -1.0 is returned as the actual_Last_Op_Time value, 
   // indicating a fault occurred.
   // 
   // 
   // 
   // ▁▁▁▁▁▁▁▁▁▁▁▁▁▁▁▁▁▁▁▁▁▁▁▁▁▁▁▁▁▁▁▁▁▁▁▁▁▁▁▁▁▁▁▁
   // 3.2.8    Detecting position faults
   // 
   // 
   // There are two types of position faults: dynamic and static. 
   // 
   // Dynamic faults occur when the valve is changing state (from open to closed or closed to open) 
   // and fails to achieve the requested position within the relevant operation time.
   // 
   // The dynamic faults are:
   // 
   //    •   Failed to open
   // 
   //    •   Failed to close
   // 
   // Static faults occur when a valve is stable in the requested state (either open or closed) and is 
   // not in the process of moving between states, and some fault occurs such that the position 
   // feedback no longer matches the requested state (e.g. the valve was correctly in the open 
   // state, and then at some point, the open feedback signal was lost without any change being 
   // made to the state of the valve by the module. Such a fault could be a power failure at the valve).
   // 
   // The static faults are:
   // 
   //    •   Failed while open
   // 
   //    •   Failed while closed
   // 
   // If the valve is not equipped with any limit switches (both CONFIG_FBK_OPEN_EN and 
   // CONFIG_FBK_CLOSED_EN are set to 0), then there are no circumstances under which any 
   // position fault can be generated (the valve is always assumed to operate correctly and be in the 
   // required position). 
   // 
   // The following table indicates the conditions under which the various alarms can be generated 
   // for the various position feedback combinations:
   // 
   //  ――――――――――――――――――――――――――――――――――――――――――
   //                    FAILED TO OPEN         FAILED TO CLOSE
   //        LIMIT SWITCH         Opening operation timer    Closing operation timer 
   //      ARRANGEMENT         expired and:                 expired and:
   //  ――――――――――――――――――――――――――――――――――――――――――
   //        No feedback
   //     CONFIG_FBK_OPEN_EN = 0     Not applicable       Not applicable
   //  CONFIG_FBK_CLOSED_EN = 0 
   // 
   //       Open feedback only
   //     CONFIG_FBK_OPEN_EN = 1   Open feedback is INACTIVE     Open feedback is ACTIVE
   //  CONFIG_FBK_CLOSED_EN = 0
   // 
   //      Closed feedback only
   //     CONFIG_FBK_OPEN_EN = 0    Closed feedback is ACTIVE     Closed feedback is INACTIVE
   //  CONFIG_FBK_CLOSED_EN = 1
   // 
   //    Open and closed feedback    Closed feedback is ACTIVE     Closed feedback is INACTIVE
   //     CONFIG_FBK_OPEN_EN = 1          OR                   OR
   //  CONFIG_FBK_CLOSED_EN = 1    Open feedback is INACTIVE     Open feedback is ACTIVE
   //  ――――――――――――――――――――――――――――――――――――――――――
   // 
   //  ――――――――――――――――――――――――――――――――――――――――――
   //                    FAILED WHILE OPEN       FAILED WHILE CLOSED
   //        LIMIT SWITCH         Opening operation timer    Closing operation timer 
   //      ARRANGEMENT         not running and:         not running and:
   //  ――――――――――――――――――――――――――――――――――――――――――
   //        No feedback
   //     CONFIG_FBK_OPEN_EN = 0     Not applicable       Not applicable
   //  CONFIG_FBK_CLOSED_EN = 0 
   // 
   //       Open feedback only
   //     CONFIG_FBK_OPEN_EN = 1   Open feedback is INACTIVE     Open feedback is ACTIVE
   //  CONFIG_FBK_CLOSED_EN = 0
   // 
   //      Closed feedback only
   //     CONFIG_FBK_OPEN_EN = 0    Closed feedback is ACTIVE     Closed feedback is INACTIVE
   //  CONFIG_FBK_CLOSED_EN = 1
   // 
   //    Open and closed feedback    Closed feedback is ACTIVE     Closed feedback is INACTIVE
   //     CONFIG_FBK_OPEN_EN = 1          OR                   OR
   //  CONFIG_FBK_CLOSED_EN = 1    Open feedback is INACTIVE     Open feedback is ACTIVE
   //  ――――――――――――――――――――――――――――――――――――――――――
   // 
   // The OR in the alarm conditions is a logical or, it covers the conditions in which both or neither 
   // limit switches are active; consider the failed to open alarm, if both limits were active, the alarm 
   // would be generated because the closed limit switch is active (irrespective of the state of the 
   // open limit). Similarly, if neither switch were active, the alarm would be generated because the 
   // open limit is inactive (irrespective of the state of the closed limit).
   // 
   // All alarms are reported as message signals, these form part of the DYNAMIC_DATA parameter 
   // UDT as follows:
   // 
   //  DATA STRUCTURE    UT31101_Dy_DevValveBi
   //  ――――――――――――――――――――――――――――――――――――――――――
   //  SIGNAL          FUNCTION                TYPE     DETAILS
   //  ――――――――――――――――――――――――――――――――――――――――――
   //  msg_FailToOpen     Valve failed to open in the specified     Bool     1 = alarm active
   //             opening operation time                0 = no alarm
   // 
   //  msg_FailToClose     Valve failed to close in the specified     Bool     1 = alarm active
   //             closing operation time               0 = no alarm
   // 
   //  msg_FailWhileOpen  Valve suffered position failure while      Bool     1 = alarm active
   //             in a static OPEN state              0 = no alarm
   // 
   //  msg_FailWhileClosed   Valve suffered position failure while      Bool     1 = alarm active
   //             in a static CLOSED state            0 = no alarm
   //  ――――――――――――――――――――――――――――――――――――――――――
END_REGION

